(* CoDeSys 2.3 export: GET_DIG_FREQ_INPUTS.EXP *)

(* POU 10_Inputs/General Parameters/Get_Dig_Freq_Inputs, ST *)
PROGRAM Get_Dig_Freq_Inputs
VAR

END_VAR
;
END_PROGRAM
